(* CODESYS project FBD_CTU.project

Project tree, tasks and I/O mapping:
  Device : CODESYS Control Win V3, 3S - Smart Software Solutions GmbH, version 3.5.15.30
    application Application
      libraries: Standard, * (System)
      task MainTask (cyclic, interval t#20ms, priority 1) calls PLC_PRG
      task VISU_TASK (cyclic, interval 100 ms, priority 31) calls VisuElems.Visu_Prg
      program PLC_PRG [FBD]
      visualisation Visualization
  text list GlobalTextList
*)

// Device/Application/PLC_PRG
PROGRAM PLC_PRG
VAR
	CTU_0: CTU;
	CTU_0_RESET: BOOL := FALSE;
	CTU_0_PV: WORD := 5;
	CTU_0_CV: WORD;
	CTU_0_Q: BOOL;
	CTU_0_CU: BOOL;
END_VAR

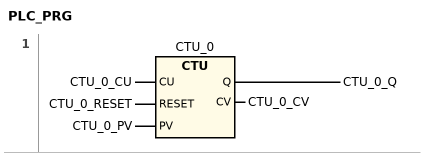
// NETWORK 1
CTU_0(CU := CTU_0_CU, RESET := CTU_0_RESET, PV := CTU_0_PV, CV => CTU_0_CV); // CTU
CTU_0_Q := CTU_0.Q;

END_PROGRAM

// Device/Application/Visualization
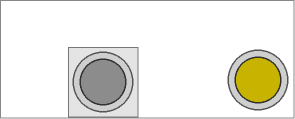
VISUALIZATION Visualization  // 295x119
    PushSwitch (68,47 70x70), variable: PLC_PRG.CTU_CU, behaviour: TOGGLE, style: Switch-PushSwitch-Gray
    Lamp1 (223,45 70x70), variable: PLC_PRG.CTU_Q, style: Lamp-Lamp1-Yellow
END_VISUALIZATION
